// TIA Portal V17 export
// export: Created 2024-09-15T12:29:43.7414594Z, ExportSetting WithDefaults, DisplayName Totally Integrated Automation Portal, DisplayVersion V17, DisplayName TIA Portal Openness, DisplayVersion V17, DisplayName TIA Portal Version Control Interface, DisplayVersion V17, DisplayName STEP 7 Professional, DisplayVersion V17, DisplayName STEP 7 Safety, DisplayVersion V17, DisplayName WinCC Professional, DisplayVersion V17
DATA_BLOCK "gtyp_SSC"   // DB13
TITLE = Global DB SSC
{ S7_Optimized_Access := 'TRUE' }
AUTHOR : A.Schaefer
VERSION : 0.0
// stored: AutoNumber true, DBAccessibleFromOPCUA true, DBAccessibleFromWebserver true, InstanceOfName typ_SSC, InstanceOfType UDT, IsOnlyStoredInLoadMemory false, IsWriteProtectedInAS false
"typ_SSC"
   // VAR RETAIN
   //    x_Start_Park_Position : Bool;
   //    x_Park_Position_Reached : Bool;
   //    x_Error : Bool;
   //    di_Pos_Centre_Horizontal : DInt := 3000;
   //    di_Pos_Centre_Vertical : DInt := 1400;
   //    di_Pos_HBW_Horizontal : DInt := 5400;
   //    di_Pos_HBW_Vertical : DInt := 950;
   //    di_Pos_Park_Horizontal : DInt := 3000;
   //    di_Pos_Park_Vertical : DInt := 200;
   //    w_Threshold_White_Red : Word := 16#25DA;
   //    w_Threshold_Red_Blue : Word := 16#3C57;
   //    Horizontal_Axis : "typ_Axis";
   //    Vertical_Axis : "typ_Axis";
   //    Workpiece : "typ_Workpiece";
   //    History { S7_SetPoint := 'True'} : Array[1..20] of "typ_History";
   // END_VAR
BEGIN
   Horizontal_Axis.i_PWM := 1000;
   Horizontal_Axis.Config.di_Pos_Soft_Switch := 5450;
   Horizontal_Axis.Config.di_Pos_Window := 25;
   Vertical_Axis.i_PWM := 1000;
   Vertical_Axis.Config.di_Pos_Soft_Switch := 3000;
   Vertical_Axis.Config.di_Pos_Window := 25;
END_DATA_BLOCK
